// Mitsubishi GX Works2 project: GX W2 L5 Ex 4 DK C   PLC: FX3G

// task Task_01 (event TRUE, interval 0, priority 31): POU_01

PROGRAM POU_01
VAR
  wProduct : INT;
  wPaintWeight : INT;
END_VAR
CASE wPaintWeight OF
0..20: wProduct := 1;
21..30: wProduct := 2;
31..40:wProduct := 3;
ELSE wProduct := 4;
END_CASE;
END_PROGRAM
